(* IEC 61131-3 sources: Lasal/CPU_5344_V01/Class/tMyBDintTODint, 1 file *)

(* ---- tMyBDintTODint.st ---- *)
(*!
<Class
	Name               = "tMyBDintTODint"
	Revision           = "0.0"
	RealtimeTask       = "false"
	CyclicTask         = "false"
	BackgroundTask     = "false"
	Sigmatek           = "false"
	OSInterface        = "false"
	HighPriority       = "false"
	Automatic          = "false"
	UpdateMode         = "Prescan"
	SharedCommandTable = "true"
	Objectsize         = "(284,180)">
	<Channels>
		<Server Name="ClassSvr" Visualized="false" Initialize="false" WriteProtected="true" Retentive="false"/>
		<Server Name="Data" Visualized="true" Initialize="false" WriteProtected="false" Retentive="false"/>
		<Client Name="cOutput" Required="true" Internal="false"/>
	</Channels>
</Class>
*)
tMyBDintTODint : CLASS
  //Servers:
	ClassSvr 	: SvrChCmd_DINT;
	Data 	: SvrCh_tMyBDint;
  //Clients:
	cOutput 	: CltCh_DINT;
  //Variables:
  //Functions:

	FUNCTION VIRTUAL GLOBAL Data::Read
		VAR_OUTPUT
			output (EAX) 	: tMyBDint;
		END_VAR;

	FUNCTION VIRTUAL GLOBAL Data::Write
		VAR_INPUT
			input (EAX) 	: tMyBDint;
		END_VAR
		VAR_OUTPUT
			result (EAX) 	: tMyBDint;
		END_VAR;
  //Tables:
	FUNCTION @STD
		VAR_OUTPUT
			ret_code	: CONFSTATES;
		END_VAR;
	FUNCTION GLOBAL TAB @CT_;
END_CLASS;

FUNCTION VIRTUAL GLOBAL tMyBDintTODint::Data::Write
	VAR_INPUT
		input (EAX) 	: tMyBDint;
	END_VAR
	VAR_OUTPUT
		result (EAX) 	: tMyBDint;
	END_VAR

  Data := Data XOR input;

  //Het significatie bit wordt ongewenst geschreven:
  //Daarom bit31 standaard altijd op '0' zetten
  Data.b31 := 0;

  cOutput := Data$dint;
  cOutput.Write(cOutput);
 	result := Data;

END_FUNCTION

FUNCTION VIRTUAL GLOBAL tMyBDintTODint::Data::Read
	VAR_OUTPUT
		output (EAX) 	: tMyBDint;
	END_VAR

  cOutput := cOutput.Read();
  Data := cOutput$tMyBDint;
	output := Data;

END_FUNCTION
